(*			
	EVERDE sp. z o.o.
	Rafał Osajda		25.10.2025		TC 4024.66
	Dodawanie meteody dla tworzenia szablownow 
*)
INTERFACE ITF_BaseCreateTemplateOfRecipe

METHOD CreateTamplateOfRecipe : BOOL
VAR_INPUT
	stTemplate				: REFERENCE TO ST_BaseRecipe;	//referencja do miejsca gdzie zostanie zapisany szablon
END_VAR
END_METHOD

END_INTERFACE

(* stored: Version 1.1.0.1
   Itf ITF_BaseCreateTemplateOfRecipe: Id {1059cad2-38ec-00a8-2713-f97371bed026}
   Method CreateTamplateOfRecipe: Id {fd74e661-f169-00b7-3578-efcb85f3e4d0} *)
